{attribute 'GeneratedUsingTerminal: EK1122-0000-0018'}
{attribute addProperty BoxType "EK1122-0000-0018"}
{attribute addProperty Id "Beckhoff_EL7xxxsub_EK1100EK1100_AB5A94672"}
{attribute addProperty CRC "291307908"}
{attribute addProperty Size "2"}
TYPE Beckhoff_EL7xxxEK1122_115D0184 EXTENDS EK1122_AB5A9467 :
STRUCT
	{attribute addProperty Name "Beckhoff_EL7xxxsub_EK1100"}
	{attribute addProperty PreviousPort "Beckhoff EL7xxxEK1122 : D"}
	Beckhoff_EL7xxxsub_EK1100 : EK1100_AB5A9467;
END_STRUCT
END_TYPE

(* stored: Version 1.2.0.0, ProductVersion 3.1.4024.9
   DUT Beckhoff_EL7xxxEK1122_115D0184: Id {b83a1c8c-b5f8-46a3-9abb-37636f4d6b7f} *)
